Staubli VAL3: onExit.pgx

public program onExit(bool x_bSave)
begin
 save:libSave()
 call set:onSave()
end
